Fanuc KAREL source: kb00107.KL

-- PROVISIONAL review KL for V940-1; original PC SHA256 eb35ab15bd240cfbdc3fd4ecef832d89b495744c8f6423fb3c3b02c9e22bd7c8
-- Incomplete behavior may be omitted. Consult companion uncertainty JSON. Do not deploy.
PROGRAM KB00107
%NOLOCKGROUP
VAR
  RESULT : BOOLEAN
-- UNRESOLVED_DECL P1 type=000106
BEGIN
  -- V9_ZERO_TABLE_METADATA_HINT layout=0001; no indexed target words; source/name/runtime held
  -- UNRESOLVED_PC offsets 5-28; opcodes 27,22,1C,27,9D,76,23
  -- UNRESOLVED_PC offsets 33-37; opcodes 7F
END KB00107
